PROGRAM MAIN
VAR
END_VAR

//Safety.bSafetyRestart 		:= IO.bInAckSignal;
//Safety.bSafetyErrorAck 		:= IO.bInAckSignal;
//Safety.bAXSafetyErrorAck 	:= IO.bInAckSignal;
//Safety.bSafetyRun 			:= TRUE;

Motion();
Toolchanger();
//TestfbSoEWrite();
//TestFBSoERead();
//TestFB_EcSetSlaveState();

END_PROGRAM

(* stored: Version 1.1.0.1, ProductVersion 3.1.4024.12
   POU MAIN: Id {824641ee-3aee-48e3-9beb-798164a31f45}, SpecialFunc None *)
